ABB RobotStudio station: standard test station_new_iteration.rsstn

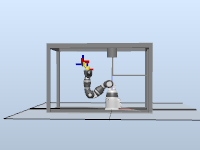
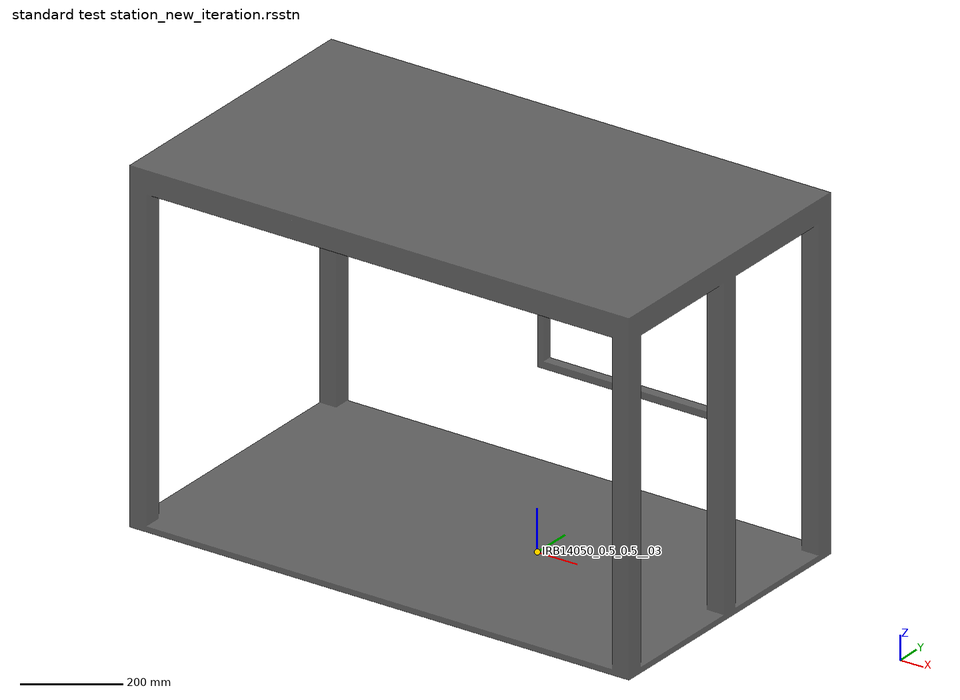
[picture v1: parts stored in the station drawn from their meshes, with robot base, taught points and paths (robot models come from the ABB library and are not in the file)]
Station standard test station (saved by RobotStudio 21.2.9526.0)
Controller Controller2
  mechanical unit ROB_1: IRB14050_0.5_0.5__03, 6 joints, base frame (0, 0, 0) mm
  mechanical unit ROB_1_7: IRB14050_0.5_0.5__03, 1 joints, base frame (0, 0, 0) mm
Layout (positions relative to the parent item):
  - IRB14050_0.5_0.5__03 [mechanism, from Robots\IRB14050_0.5_0.5__03.rslib] at (0, 0, 0) mm; joint values [0, -2.3562, 0, 0.7854, 0, 0, 0] (rad or m)
  - roof [part], size 1180 x 680 x 12 mm
  - horizontal_pole_1 [part], size 1180 x 40 x 40 mm
  - horizontal_pole_2 [part], size 1180 x 40 x 40 mm
  - horizontal_pole_3 [part], size 40 x 600 x 40 mm
  - horizontal_pole_4 [part], size 40 x 600 x 40 mm
  - cylinder [part], size 120 x 119.8 x 120 mm
  - vertical_pole_1 [part], size 40 x 40 x 743 mm
  - vertical_pole_2 [part], size 40 x 40 x 743 mm
  - middle_vertical_pole [part], size 40 x 40 x 743 mm
  - vertical_pole_3 [part], size 40 x 40 x 743 mm
  - vertical_pole_4 [part], size 40 x 40 x 743 mm
  - sender_pole [part], size 430 x 22.5 x 15 mm
  - linear_actuator [part], size 15 x 22.5 x 208 mm
  - floor [part], size 1180 x 680 x 12 mm
  - IRB14050_new_iteration_tool [mechanism, from Robot Studio\IRB14050_new_iteration_tool.rslib] at (-298.19, 0, 479.01) mm
Attachment: IRB14050_new_iteration_tool is attached to IRB14050_0.5_0.5__03 / Link7
Collision set robot_cylinder: IRB14050_0.5_0.5__03 against cylinder, near miss 0 m
Collision set robot_linear_act: IRB14050_0.5_0.5__03 against linear_actuator, near miss 0 m
Collision set robot_horizontal_1: IRB14050_0.5_0.5__03 against horizontal_pole_1, near miss 0 m
Collision set robot_horizontal_2: IRB14050_0.5_0.5__03 against horizontal_pole_2, near miss 0 m
Collision set robot_middle_pole: IRB14050_0.5_0.5__03 against middle_vertical_pole, near miss 0 m
Collision set robot_roof: IRB14050_0.5_0.5__03 against roof, near miss 0 m
Collision set robot_sender_pole: IRB14050_0.5_0.5__03 against sender_pole, near miss 0 m
Collision set robot_horizontal_3: IRB14050_0.5_0.5__03 against horizontal_pole_3, near miss 0 m
Collision set robot_horizontal_4: IRB14050_0.5_0.5__03 against horizontal_pole_4, near miss 0 m
Collision set robot_vertical_1: IRB14050_0.5_0.5__03 against vertical_pole_1, near miss 0 m
Collision set robot_vertical_2: IRB14050_0.5_0.5__03 against vertical_pole_2, near miss 0 m
Collision set robot_vertical_3: IRB14050_0.5_0.5__03 against vertical_pole_3, near miss 0 m
Collision set robot_vertical_4: IRB14050_0.5_0.5__03 against vertical_pole_4, near miss 0 m
Collision set tool_cylinder: IRB14050_new_iteration_tool against cylinder, near miss 0 m
Collision set tool_floor: IRB14050_new_iteration_tool against floor, near miss 0 m
Collision set tool_horizontal_pole_1: IRB14050_new_iteration_tool against horizontal_pole_1, near miss 0 m
Collision set tool_horizontal_pole_2: IRB14050_new_iteration_tool against horizontal_pole_2, near miss 0 m
Collision set tool_horizontal_pole_3: IRB14050_new_iteration_tool against horizontal_pole_3, near miss 0 m
Collision set tool_horizontal_pole_4: IRB14050_new_iteration_tool against horizontal_pole_4, near miss 0 m
Collision set tool_linear_actuator: IRB14050_new_iteration_tool against linear_actuator, near miss 0 m
Collision set tool_middle_vertical_pole: IRB14050_new_iteration_tool against middle_vertical_pole, near miss 0 m
Collision set tool_roof: IRB14050_new_iteration_tool against roof, near miss 0 m
Collision set tool_sender_pole: IRB14050_new_iteration_tool against sender_pole, near miss 0 m
Collision set tool_vertical_pole_1: IRB14050_new_iteration_tool against vertical_pole_1, near miss 0 m
Collision set tool_vertical_pole_2: IRB14050_new_iteration_tool against vertical_pole_2, near miss 0 m
Collision set tool_vertical_pole_3: IRB14050_new_iteration_tool against vertical_pole_3, near miss 0 m
Collision set tool_vertical_pole_4: IRB14050_new_iteration_tool against vertical_pole_4, near miss 0 m
Targets, tools, work objects and paths stored in the station, written as RAPID:
! task T_ROB1
MODULE CalibData
  PERS tooldata tcp_laser:=[TRUE,[[-51.474,3.9,86.55],[1,0,0,0]],[0.1,[-27.92,-2.835,45.984],[1,0,0,0],0,0,0]];
  PERS tooldata tcp_calibration:=[TRUE,[[-61.474,-13.499,62.227],[0.707106781,0,-0.707106781,0]],[0.1,[-27.92,-2.835,45.984],[1,0,0,0],0,0,0]];
  PERS tooldata tcp_antenna:=[TRUE,[[-53.974,33.75,100.5],[1,0,0,0]],[0.1,[-27.92,-2.835,45.984],[1,0,0,0],0,0,0]];
ENDMODULE

